INTERFACE ITransport EXTENDS ZApplication.IUnit

END_INTERFACE

(* stored: Version 1.1.0.1
   Itf ITransport: Id {15a9683e-0e83-4913-9964-5a1ff7ef54ae} *)
